// TIA Portal V15.1 export
// export: Created 2020-06-12T07:35:52.8193359Z, ExportSetting None, DisplayName Totally Integrated Automation Portal, DisplayVersion V15.1, DisplayName TIA Portal Openness, DisplayVersion V15.1, DisplayName STEP 7 Professional, DisplayVersion V15.1, DisplayName STEP 7 Safety, DisplayVersion V15.1, DisplayName WinCC Advanced, DisplayVersion V15.1
FUNCTION "MELT_Subsys" : Void   // FC174, FBD
{ S7_Optimized_Access := 'TRUE' }
// stored: SetENOAutomatically False
   VAR_TEMP
      tBool : Bool;
      _act_am : Real;
      _recipe_set : Real;
      tGasPressNorm : Real;
      _melt_gas_on : Bool;
      _melt_gas_mode : Int;
      tStartSlagToLoad : Bool;
      tMeltSlagToLoad : Bool;
      tRate : Real;
      tDuration : Real;
      tSlagDosTime : LReal;
      tSlagDoseTimeout : Bool;
      tEndMelt : Bool;
      tGasPressHT : Real;
      tBaseWeight : Real;
      tDedCmdOff : Bool;
      tReqVentOFF : Bool;
      tVentOffTime : Time;
   END_VAR
   VAR_TEMP   // added for the SCL form of the ladder/FBD networks
      _w1 : Bool;
      _w2 : Bool;
      _w3 : Bool;
   END_VAR
BEGIN

REGION Network 1: End melt flag
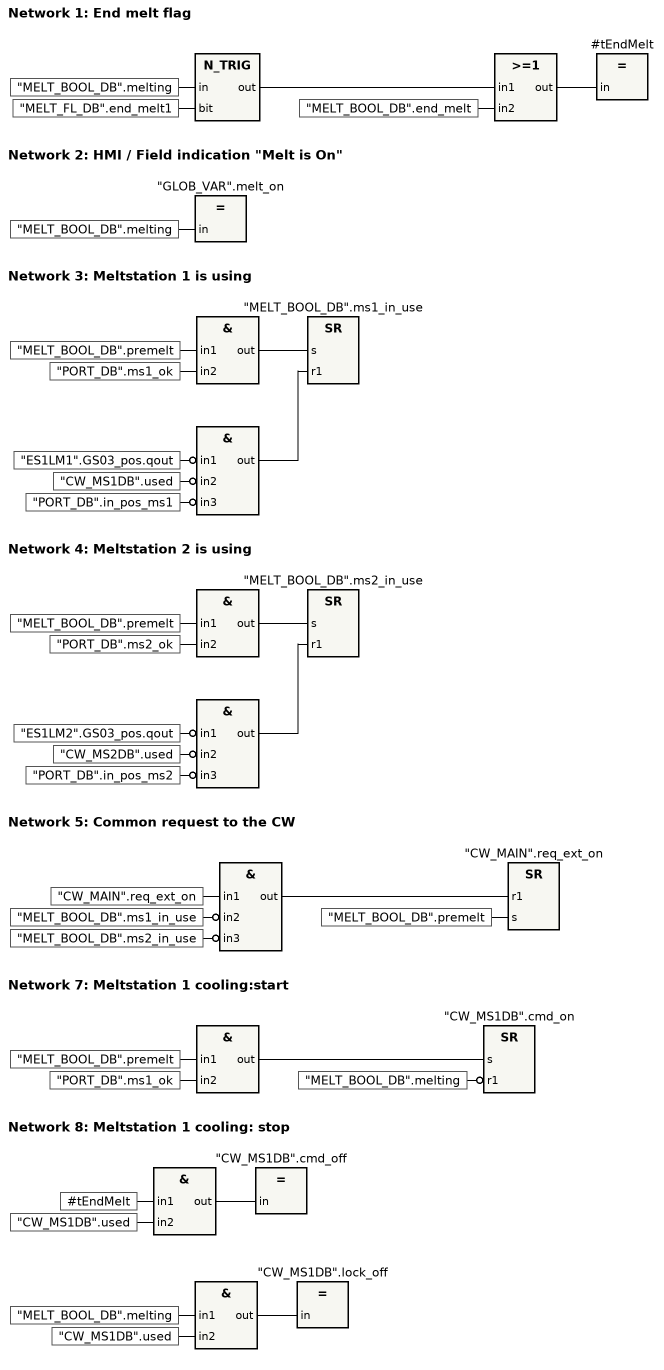
   #_w1 := NOT "MELT_BOOL_DB".melting AND "MELT_FL_DB".end_melt1;   // falling edge
   "MELT_FL_DB".end_melt1 := "MELT_BOOL_DB".melting;
   #tEndMelt := #_w1 OR "MELT_BOOL_DB".end_melt;
END_REGION

REGION Network 2: HMI / Field indication "Melt is On"
   "GLOB_VAR".melt_on := "MELT_BOOL_DB".melting;
END_REGION

REGION Network 3: Meltstation 1 is using
   IF "MELT_BOOL_DB".premelt AND "PORT_DB".ms1_ok THEN
       "MELT_BOOL_DB".ms1_in_use := TRUE;   // SR flip-flop
   END_IF;
   IF NOT "ES1LM1".GS03_pos.qout AND NOT "CW_MS1DB".used AND NOT "PORT_DB".in_pos_ms1 THEN
       "MELT_BOOL_DB".ms1_in_use := FALSE;
   END_IF;
END_REGION

REGION Network 4: Meltstation 2 is using
   IF "MELT_BOOL_DB".premelt AND "PORT_DB".ms2_ok THEN
       "MELT_BOOL_DB".ms2_in_use := TRUE;   // SR flip-flop
   END_IF;
   IF NOT "ES1LM2".GS03_pos.qout AND NOT "CW_MS2DB".used AND NOT "PORT_DB".in_pos_ms2 THEN
       "MELT_BOOL_DB".ms2_in_use := FALSE;
   END_IF;
END_REGION

REGION Network 5: Common request to the CW
   #_w1 := "CW_MAIN".req_ext_on AND NOT "MELT_BOOL_DB".ms1_in_use AND NOT "MELT_BOOL_DB".ms2_in_use;
   IF "MELT_BOOL_DB".premelt THEN
       "CW_MAIN".req_ext_on := TRUE;   // SR flip-flop
   END_IF;
   IF #_w1 THEN "CW_MAIN".req_ext_on := FALSE; END_IF;
END_REGION

REGION Network 6: [Cooling Water System]
END_REGION

REGION Network 7: Meltstation 1 cooling:start
   IF "MELT_BOOL_DB".premelt AND "PORT_DB".ms1_ok THEN
       "CW_MS1DB".cmd_on := TRUE;   // SR flip-flop
   END_IF;
   IF NOT "MELT_BOOL_DB".melting THEN "CW_MS1DB".cmd_on := FALSE; END_IF;
END_REGION

REGION Network 8: Meltstation 1 cooling: stop
   "CW_MS1DB".cmd_off := #tEndMelt AND "CW_MS1DB".used;
   "CW_MS1DB".lock_off := "MELT_BOOL_DB".melting AND "CW_MS1DB".used;
END_REGION

REGION Network 9: Meltstation 1 cooling: control the flow
   // We use always flow control
   // NB That's good place for that instruction, becuase we can add any process-related variable here if needed
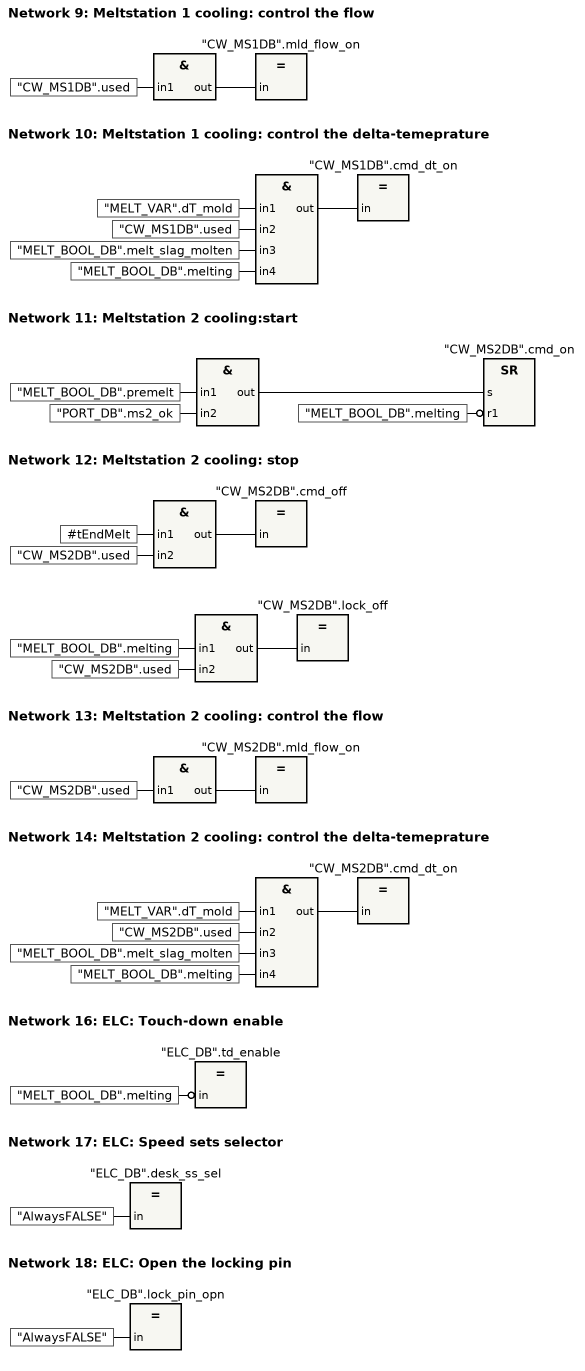
   "CW_MS1DB".mld_flow_on := "CW_MS1DB".used;
END_REGION

REGION Network 10: Meltstation 1 cooling: control the delta-temeprature
   "CW_MS1DB".cmd_dt_on := "MELT_VAR".dT_mold AND "CW_MS1DB".used AND "MELT_BOOL_DB".melt_slag_molten AND "MELT_BOOL_DB".melting;
END_REGION

REGION Network 11: Meltstation 2 cooling:start
   IF "MELT_BOOL_DB".premelt AND "PORT_DB".ms2_ok THEN
       "CW_MS2DB".cmd_on := TRUE;   // SR flip-flop
   END_IF;
   IF NOT "MELT_BOOL_DB".melting THEN "CW_MS2DB".cmd_on := FALSE; END_IF;
END_REGION

REGION Network 12: Meltstation 2 cooling: stop
   "CW_MS2DB".cmd_off := #tEndMelt AND "CW_MS2DB".used;
   "CW_MS2DB".lock_off := "MELT_BOOL_DB".melting AND "CW_MS2DB".used;
END_REGION

REGION Network 13: Meltstation 2 cooling: control the flow
   "CW_MS2DB".mld_flow_on := "CW_MS2DB".used;
END_REGION

REGION Network 14: Meltstation 2 cooling: control the delta-temeprature
   "CW_MS2DB".cmd_dt_on := "MELT_VAR".dT_mold AND "CW_MS2DB".used AND "MELT_BOOL_DB".melt_slag_molten AND "MELT_BOOL_DB".melting;
END_REGION

REGION Network 15: [Plant]
END_REGION

REGION Network 16: ELC: Touch-down enable
   "ELC_DB".td_enable := NOT "MELT_BOOL_DB".melting;
END_REGION

REGION Network 17: ELC: Speed sets selector
   "ELC_DB".desk_ss_sel := "AlwaysFALSE";
END_REGION

REGION Network 18: ELC: Open the locking pin
   // NB: WTF?
   "ELC_DB".lock_pin_opn := "AlwaysFALSE";
END_REGION

REGION Network 19: ELC-XY lock
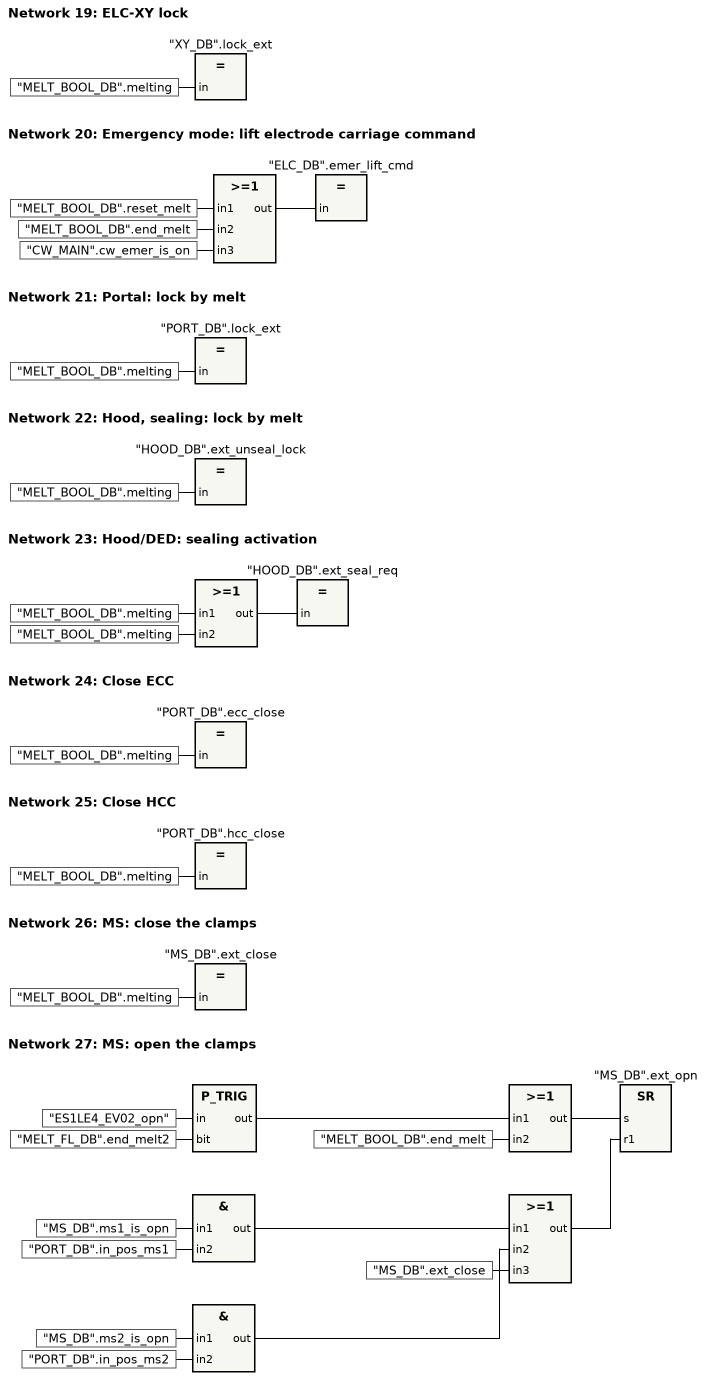
   "XY_DB".lock_ext := "MELT_BOOL_DB".melting;
END_REGION

REGION Network 20: Emergency mode: lift electrode carriage command
   "ELC_DB".emer_lift_cmd := "MELT_BOOL_DB".reset_melt OR "MELT_BOOL_DB".end_melt OR "CW_MAIN".cw_emer_is_on;
END_REGION

REGION Network 21: Portal: lock by melt
   "PORT_DB".lock_ext := "MELT_BOOL_DB".melting;
END_REGION

REGION Network 22: Hood, sealing: lock by melt
   "HOOD_DB".ext_unseal_lock := "MELT_BOOL_DB".melting;
END_REGION

REGION Network 23: Hood/DED: sealing activation
   "HOOD_DB".ext_seal_req := "MELT_BOOL_DB".melting OR "MELT_BOOL_DB".melting;
END_REGION

REGION Network 24: Close ECC
   "PORT_DB".ecc_close := "MELT_BOOL_DB".melting;
END_REGION

REGION Network 25: Close HCC
   "PORT_DB".hcc_close := "MELT_BOOL_DB".melting;
END_REGION

REGION Network 26: MS: close the clamps
   "MS_DB".ext_close := "MELT_BOOL_DB".melting;
END_REGION

REGION Network 27: MS: open the clamps
   #_w1 := "ES1LE4_EV02_opn" AND NOT "MELT_FL_DB".end_melt2;   // rising edge
   "MELT_FL_DB".end_melt2 := "ES1LE4_EV02_opn";
   IF #_w1 OR "MELT_BOOL_DB".end_melt THEN
       "MS_DB".ext_opn := TRUE;   // SR flip-flop
   END_IF;
   IF ("MS_DB".ms1_is_opn AND "PORT_DB".in_pos_ms1) OR ("MS_DB".ms2_is_opn AND "PORT_DB".in_pos_ms2) OR "MS_DB".ext_close THEN
       "MS_DB".ext_opn := FALSE;
   END_IF;
END_REGION

REGION Network 28: [Gas feeding]
END_REGION

REGION Network 29: Reset volume counters before melt
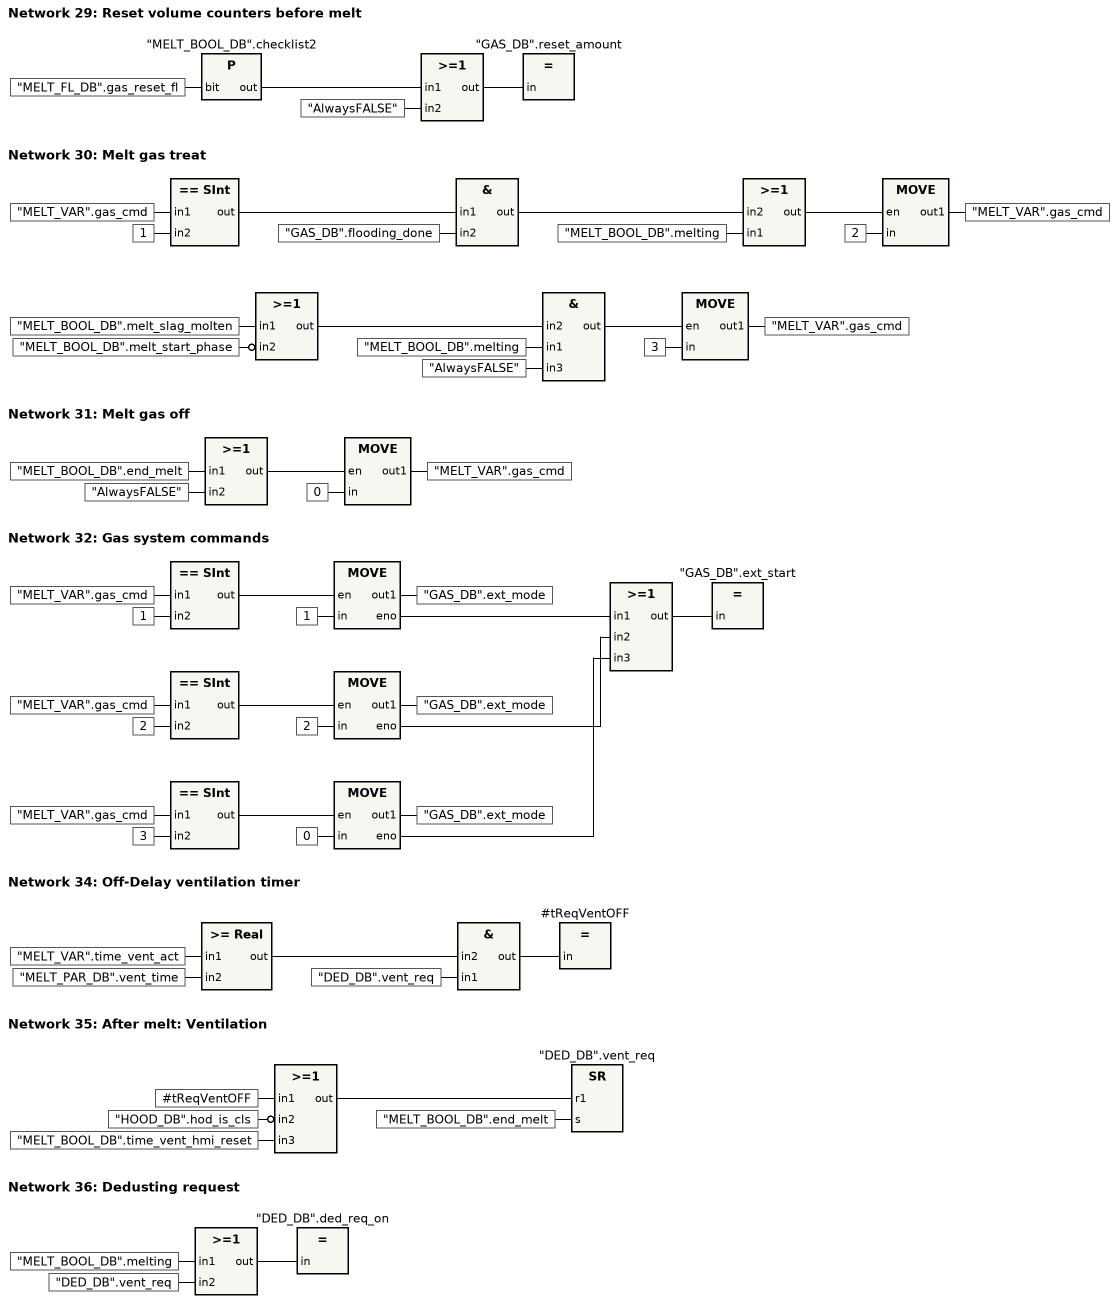
   #_w1 := "MELT_BOOL_DB".checklist2 AND NOT "MELT_FL_DB".gas_reset_fl;   // rising edge of "MELT_BOOL_DB".checklist2
   "MELT_FL_DB".gas_reset_fl := "MELT_BOOL_DB".checklist2;
   "GAS_DB".reset_amount := #_w1 OR "AlwaysFALSE";
END_REGION

REGION Network 30: Melt gas treat
   // NB: The constant flow mode during melt is not needed - it is enought "pressure limit" mode
   IF (("MELT_VAR".gas_cmd = 1) AND "GAS_DB".flooding_done) OR "MELT_BOOL_DB".melting THEN
       "MELT_VAR".gas_cmd := 2;
   END_IF;
   IF ("MELT_BOOL_DB".melt_slag_molten OR NOT "MELT_BOOL_DB".melt_start_phase) AND "MELT_BOOL_DB".melting AND "AlwaysFALSE" THEN
       "MELT_VAR".gas_cmd := 3;
   END_IF;
END_REGION

REGION Network 31: Melt gas off
   IF "MELT_BOOL_DB".end_melt OR "AlwaysFALSE" THEN "MELT_VAR".gas_cmd := 0; END_IF;
END_REGION

REGION Network 32: Gas system commands
   #_w1 := "MELT_VAR".gas_cmd = 1;
   IF #_w1 THEN "GAS_DB".ext_mode := 1; END_IF;
   #_w2 := "MELT_VAR".gas_cmd = 2;
   IF #_w2 THEN "GAS_DB".ext_mode := 2; END_IF;
   #_w3 := "MELT_VAR".gas_cmd = 3;
   IF #_w3 THEN "GAS_DB".ext_mode := 0; END_IF;
   "GAS_DB".ext_start := #_w1 OR #_w2 OR #_w3;
END_REGION

REGION Network 33: [Dedusting]
END_REGION

REGION Network 34: Off-Delay ventilation timer
   #tReqVentOFF := ("MELT_VAR".time_vent_act >= "MELT_PAR_DB".vent_time) AND "DED_DB".vent_req;
END_REGION

REGION Network 35: After melt: Ventilation
   IF "MELT_BOOL_DB".end_melt THEN
       "DED_DB".vent_req := TRUE;   // SR flip-flop
   END_IF;
   IF #tReqVentOFF OR NOT "HOOD_DB".hod_is_cls OR "MELT_BOOL_DB".time_vent_hmi_reset THEN
       "DED_DB".vent_req := FALSE;
   END_IF;
END_REGION

REGION Network 36: Dedusting request
   "DED_DB".ded_req_on := "MELT_BOOL_DB".melting OR "DED_DB".vent_req;
END_REGION

REGION Network 37: [[END]]
END_REGION
END_FUNCTION
